// TIA Portal V17 export
// export: Created 2025-03-07T09:17:41.1977773Z, ExportSetting WithDefaults, DisplayName Totally Integrated Automation Portal, DisplayVersion V17 Update 8, DisplayName TIA Portal Openness, DisplayVersion V17 Update 8, DisplayName TIA Portal Version Control Interface, DisplayVersion V17, DisplayName SINAMICS Startdrive Advanced, DisplayVersion V17 SP2, DisplayName SINAMICS Startdrive G110M, G120, G120C, G120D, G120P, G115D, DisplayVersion V17 SP2, DisplayName SINAMICS Startdrive G130, G150, S120, S150, SINAMICS MV, S210, DisplayVersion V17 SP2, DisplayName STEP 7 Professional, DisplayVersion V17 Update 8, DisplayName SINUMERIK ONE STEP 7 Toolbox, DisplayVersion V17 Update 12, DisplayName SINUMERIK 840D sl STEP 7 Toolbox, DisplayVersion V17 Update 12, DisplayName STEP 7 Safety, DisplayVersion V17 Update 6, DisplayName WinCC Advanced, DisplayVersion V17 Update 8
FUNCTION "FC2027_INCREMENTAL_MODE_MG2" : Void   // FC2027, LAD
{ S7_Optimized_Access := 'FALSE' }
AUTHOR : ETXETAR
VERSION : 1.0
// stored: AutoNumber false, IsIECCheckEnabled false, SetENOAutomatically false, UDAEnableTagReadback false
   VAR CONSTANT
      FC_NUMBER : DInt := 2027;
   END_VAR
   VAR_TEMP   // added for the SCL form of the ladder/FBD networks
      _w1 : Bool;
      _w2 : Bool;
   END_VAR
BEGIN

REGION Network 1: GENERAL CONDITIONS
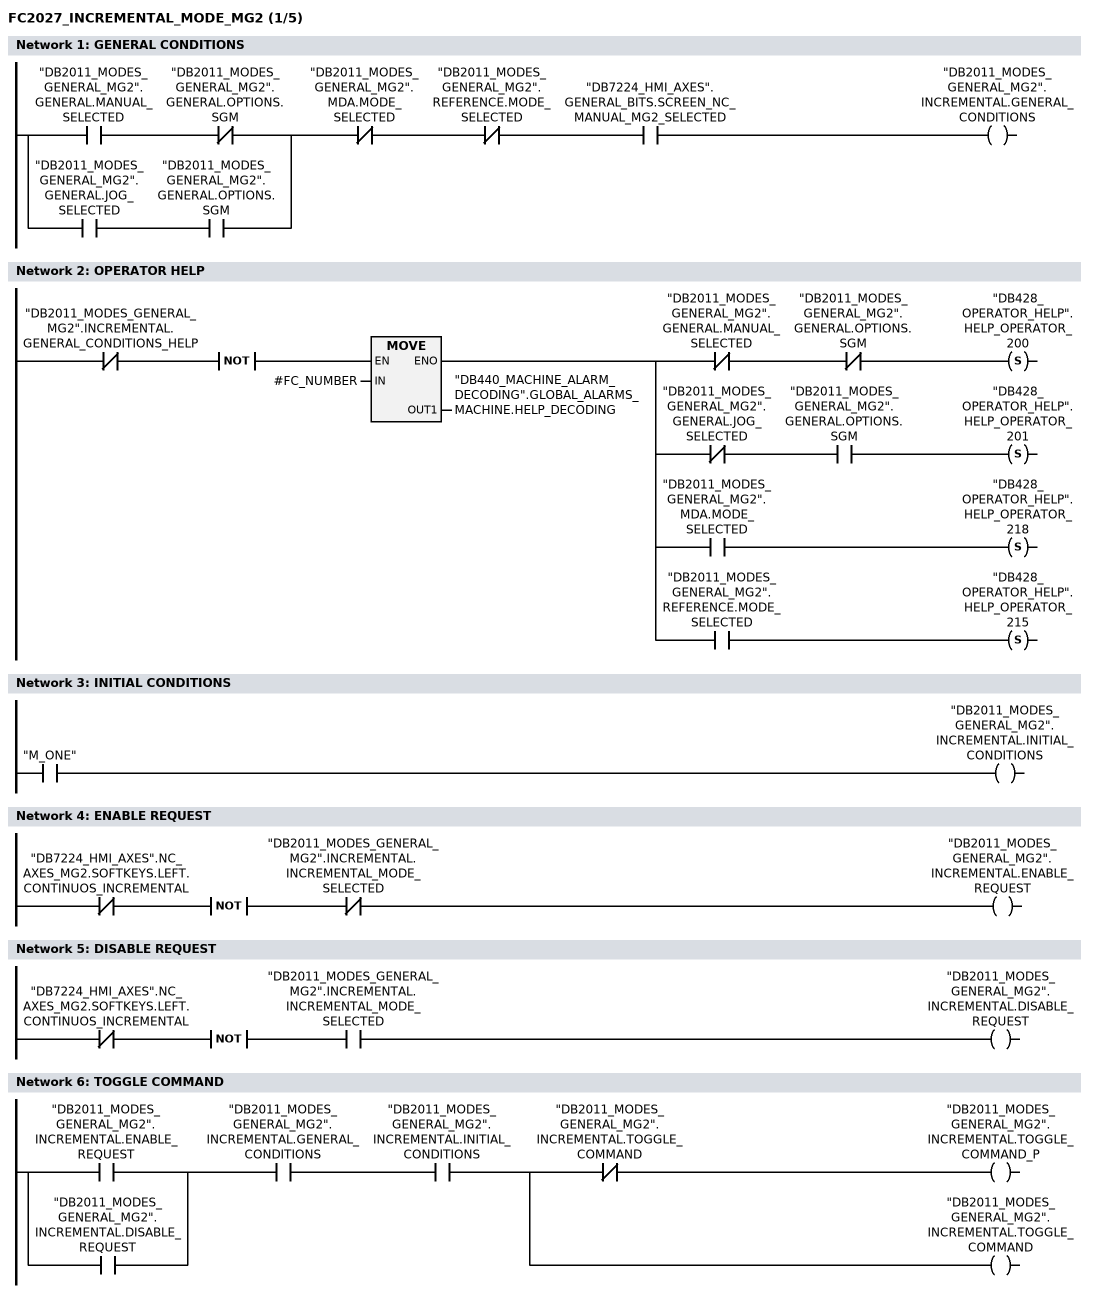
   RUNG wire#powerrail
      Contact( "DB2011_MODES_GENERAL_MG2".GENERAL.MANUAL_SELECTED )
      I_Contact( "DB2011_MODES_GENERAL_MG2".GENERAL.OPTIONS.SGM )
      wire#w1
      I_Contact( "DB2011_MODES_GENERAL_MG2".MDA.MODE_SELECTED )
      I_Contact( "DB2011_MODES_GENERAL_MG2".REFERENCE.MODE_SELECTED )
      Contact( "DB7224_HMI_AXES".GENERAL_BITS.SCREEN_NC_MANUAL_MG2_SELECTED )
      Coil( "DB2011_MODES_GENERAL_MG2".INCREMENTAL.GENERAL_CONDITIONS )
   END_RUNG
   RUNG wire#powerrail
      Contact( "DB2011_MODES_GENERAL_MG2".GENERAL.JOG_SELECTED )
      Contact( "DB2011_MODES_GENERAL_MG2".GENERAL.OPTIONS.SGM )
   END_RUNG wire#w1
   // the same network as SCL:
   "DB2011_MODES_GENERAL_MG2".INCREMENTAL.GENERAL_CONDITIONS := (("DB2011_MODES_GENERAL_MG2".GENERAL.MANUAL_SELECTED AND NOT "DB2011_MODES_GENERAL_MG2".GENERAL.OPTIONS.SGM) OR ("DB2011_MODES_GENERAL_MG2".GENERAL.JOG_SELECTED AND "DB2011_MODES_GENERAL_MG2".GENERAL.OPTIONS.SGM)) AND NOT "DB2011_MODES_GENERAL_MG2".MDA.MODE_SELECTED AND NOT "DB2011_MODES_GENERAL_MG2".REFERENCE.MODE_SELECTED AND "DB7224_HMI_AXES".GENERAL_BITS.SCREEN_NC_MANUAL_MG2_SELECTED;
END_REGION

REGION Network 2: OPERATOR HELP
   RUNG wire#powerrail
      I_Contact( "DB2011_MODES_GENERAL_MG2".INCREMENTAL.GENERAL_CONDITIONS_HELP )
      Not()
      { S7_GenerateENO := "TRUE" } Move(in := #FC_NUMBER, out1 => "DB440_MACHINE_ALARM_DECODING".GLOBAL_ALARMS_MACHINE.HELP_DECODING)
      wire#w1
      I_Contact( "DB2011_MODES_GENERAL_MG2".GENERAL.MANUAL_SELECTED )
      I_Contact( "DB2011_MODES_GENERAL_MG2".GENERAL.OPTIONS.SGM )
      S_Coil( "DB428_OPERATOR_HELP".HELP_OPERATOR_200 )
   END_RUNG
   RUNG wire#w1
      I_Contact( "DB2011_MODES_GENERAL_MG2".GENERAL.JOG_SELECTED )
      Contact( "DB2011_MODES_GENERAL_MG2".GENERAL.OPTIONS.SGM )
      S_Coil( "DB428_OPERATOR_HELP".HELP_OPERATOR_201 )
   END_RUNG
   RUNG wire#w1
      Contact( "DB2011_MODES_GENERAL_MG2".MDA.MODE_SELECTED )
      S_Coil( "DB428_OPERATOR_HELP".HELP_OPERATOR_218 )
   END_RUNG
   RUNG wire#w1
      Contact( "DB2011_MODES_GENERAL_MG2".REFERENCE.MODE_SELECTED )
      S_Coil( "DB428_OPERATOR_HELP".HELP_OPERATOR_215 )
   END_RUNG
   // the same network as SCL:
   // ENO of a box is taken as its EN; it also drops when the box reports an error
   #_w1 := NOT (NOT "DB2011_MODES_GENERAL_MG2".INCREMENTAL.GENERAL_CONDITIONS_HELP);
   IF #_w1 THEN "DB440_MACHINE_ALARM_DECODING".GLOBAL_ALARMS_MACHINE.HELP_DECODING := #FC_NUMBER; END_IF;
   IF #_w1 AND NOT "DB2011_MODES_GENERAL_MG2".GENERAL.MANUAL_SELECTED AND NOT "DB2011_MODES_GENERAL_MG2".GENERAL.OPTIONS.SGM THEN
       "DB428_OPERATOR_HELP".HELP_OPERATOR_200 := TRUE;
   END_IF;
   IF #_w1 AND NOT "DB2011_MODES_GENERAL_MG2".GENERAL.JOG_SELECTED AND "DB2011_MODES_GENERAL_MG2".GENERAL.OPTIONS.SGM THEN
       "DB428_OPERATOR_HELP".HELP_OPERATOR_201 := TRUE;
   END_IF;
   IF #_w1 AND "DB2011_MODES_GENERAL_MG2".MDA.MODE_SELECTED THEN
       "DB428_OPERATOR_HELP".HELP_OPERATOR_218 := TRUE;
   END_IF;
   IF #_w1 AND "DB2011_MODES_GENERAL_MG2".REFERENCE.MODE_SELECTED THEN
       "DB428_OPERATOR_HELP".HELP_OPERATOR_215 := TRUE;
   END_IF;
END_REGION

REGION Network 3: INITIAL CONDITIONS
   RUNG wire#powerrail
      Contact( "M_ONE" )
      Coil( "DB2011_MODES_GENERAL_MG2".INCREMENTAL.INITIAL_CONDITIONS )
   END_RUNG
   // the same network as SCL:
   "DB2011_MODES_GENERAL_MG2".INCREMENTAL.INITIAL_CONDITIONS := "M_ONE";
END_REGION

REGION Network 4: ENABLE REQUEST
   RUNG wire#powerrail
      I_Contact( "DB7224_HMI_AXES".NC_AXES_MG2.SOFTKEYS.LEFT.CONTINUOS_INCREMENTAL )
      Not()
      I_Contact( "DB2011_MODES_GENERAL_MG2".INCREMENTAL.INCREMENTAL_MODE_SELECTED )
      Coil( "DB2011_MODES_GENERAL_MG2".INCREMENTAL.ENABLE_REQUEST )
   END_RUNG
   // the same network as SCL:
   "DB2011_MODES_GENERAL_MG2".INCREMENTAL.ENABLE_REQUEST := NOT (NOT "DB7224_HMI_AXES".NC_AXES_MG2.SOFTKEYS.LEFT.CONTINUOS_INCREMENTAL) AND NOT "DB2011_MODES_GENERAL_MG2".INCREMENTAL.INCREMENTAL_MODE_SELECTED;
END_REGION

REGION Network 5: DISABLE REQUEST
   RUNG wire#powerrail
      I_Contact( "DB7224_HMI_AXES".NC_AXES_MG2.SOFTKEYS.LEFT.CONTINUOS_INCREMENTAL )
      Not()
      Contact( "DB2011_MODES_GENERAL_MG2".INCREMENTAL.INCREMENTAL_MODE_SELECTED )
      Coil( "DB2011_MODES_GENERAL_MG2".INCREMENTAL.DISABLE_REQUEST )
   END_RUNG
   // the same network as SCL:
   "DB2011_MODES_GENERAL_MG2".INCREMENTAL.DISABLE_REQUEST := NOT (NOT "DB7224_HMI_AXES".NC_AXES_MG2.SOFTKEYS.LEFT.CONTINUOS_INCREMENTAL) AND "DB2011_MODES_GENERAL_MG2".INCREMENTAL.INCREMENTAL_MODE_SELECTED;
END_REGION

REGION Network 6: TOGGLE COMMAND
   RUNG wire#powerrail
      Contact( "DB2011_MODES_GENERAL_MG2".INCREMENTAL.ENABLE_REQUEST )
      wire#w1
      Contact( "DB2011_MODES_GENERAL_MG2".INCREMENTAL.GENERAL_CONDITIONS )
      Contact( "DB2011_MODES_GENERAL_MG2".INCREMENTAL.INITIAL_CONDITIONS )
      wire#w2
      I_Contact( "DB2011_MODES_GENERAL_MG2".INCREMENTAL.TOGGLE_COMMAND )
      Coil( "DB2011_MODES_GENERAL_MG2".INCREMENTAL.TOGGLE_COMMAND_P )
   END_RUNG
   RUNG wire#powerrail
      Contact( "DB2011_MODES_GENERAL_MG2".INCREMENTAL.DISABLE_REQUEST )
   END_RUNG wire#w1
   RUNG wire#w2
      Coil( "DB2011_MODES_GENERAL_MG2".INCREMENTAL.TOGGLE_COMMAND )
   END_RUNG
   // the same network as SCL:
   #_w1 := ("DB2011_MODES_GENERAL_MG2".INCREMENTAL.ENABLE_REQUEST OR "DB2011_MODES_GENERAL_MG2".INCREMENTAL.DISABLE_REQUEST) AND "DB2011_MODES_GENERAL_MG2".INCREMENTAL.GENERAL_CONDITIONS AND "DB2011_MODES_GENERAL_MG2".INCREMENTAL.INITIAL_CONDITIONS;
   "DB2011_MODES_GENERAL_MG2".INCREMENTAL.TOGGLE_COMMAND_P := #_w1 AND NOT "DB2011_MODES_GENERAL_MG2".INCREMENTAL.TOGGLE_COMMAND;
   "DB2011_MODES_GENERAL_MG2".INCREMENTAL.TOGGLE_COMMAND := #_w1;
END_REGION

REGION Network 7: INCREMENTAL MODE SELECTED
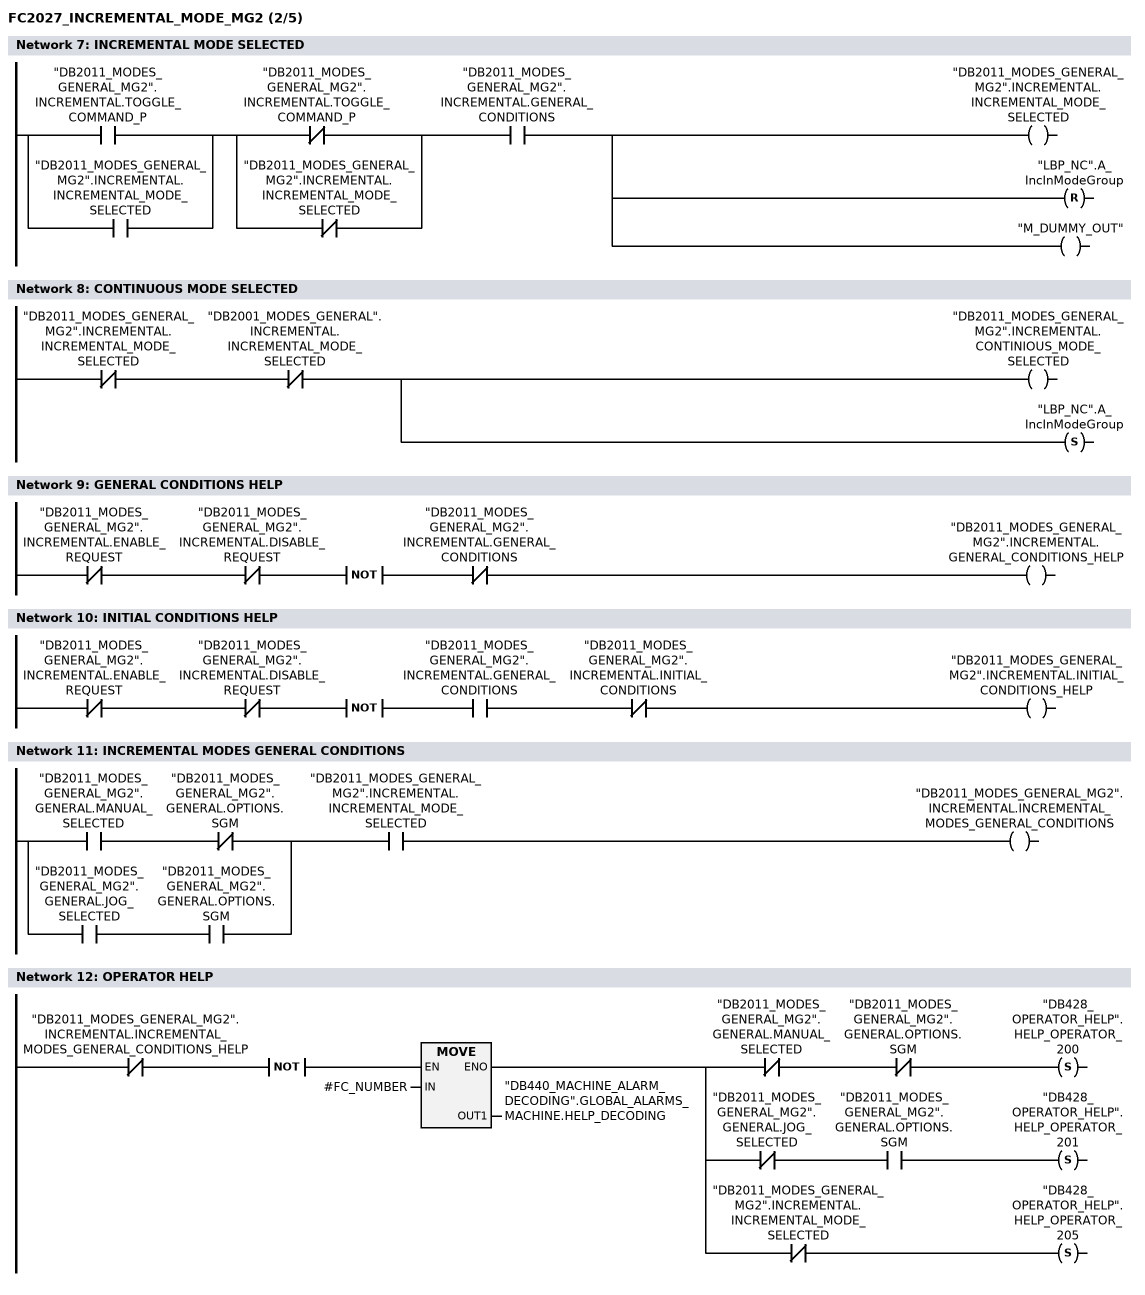
   RUNG wire#powerrail
      Contact( "DB2011_MODES_GENERAL_MG2".INCREMENTAL.TOGGLE_COMMAND_P )
      wire#w1
      I_Contact( "DB2011_MODES_GENERAL_MG2".INCREMENTAL.TOGGLE_COMMAND_P )
      wire#w2
      Contact( "DB2011_MODES_GENERAL_MG2".INCREMENTAL.GENERAL_CONDITIONS )
      wire#w3
      Coil( "DB2011_MODES_GENERAL_MG2".INCREMENTAL.INCREMENTAL_MODE_SELECTED )
   END_RUNG
   RUNG wire#powerrail
      Contact( "DB2011_MODES_GENERAL_MG2".INCREMENTAL.INCREMENTAL_MODE_SELECTED )
   END_RUNG wire#w1
   RUNG wire#w1
      I_Contact( "DB2011_MODES_GENERAL_MG2".INCREMENTAL.INCREMENTAL_MODE_SELECTED )
   END_RUNG wire#w2
   RUNG wire#w3
      R_Coil( "LBP_NC".A_IncInModeGroup )
   END_RUNG
   RUNG wire#w3
      Coil( "M_DUMMY_OUT" )
   END_RUNG
   // the same network as SCL:
   "DB2011_MODES_GENERAL_MG2".INCREMENTAL.INCREMENTAL_MODE_SELECTED := ("DB2011_MODES_GENERAL_MG2".INCREMENTAL.TOGGLE_COMMAND_P OR "DB2011_MODES_GENERAL_MG2".INCREMENTAL.INCREMENTAL_MODE_SELECTED) AND (NOT "DB2011_MODES_GENERAL_MG2".INCREMENTAL.TOGGLE_COMMAND_P OR NOT "DB2011_MODES_GENERAL_MG2".INCREMENTAL.INCREMENTAL_MODE_SELECTED) AND "DB2011_MODES_GENERAL_MG2".INCREMENTAL.GENERAL_CONDITIONS;
   IF "DB2011_MODES_GENERAL_MG2".INCREMENTAL.INCREMENTAL_MODE_SELECTED THEN
       "LBP_NC".A_IncInModeGroup := FALSE;
   END_IF;
   "M_DUMMY_OUT" := "DB2011_MODES_GENERAL_MG2".INCREMENTAL.INCREMENTAL_MODE_SELECTED;
END_REGION

REGION Network 8: CONTINUOUS MODE SELECTED
   RUNG wire#powerrail
      I_Contact( "DB2011_MODES_GENERAL_MG2".INCREMENTAL.INCREMENTAL_MODE_SELECTED )
      I_Contact( "DB2001_MODES_GENERAL".INCREMENTAL.INCREMENTAL_MODE_SELECTED )
      wire#w1
      Coil( "DB2011_MODES_GENERAL_MG2".INCREMENTAL.CONTINIOUS_MODE_SELECTED )
   END_RUNG
   RUNG wire#w1
      S_Coil( "LBP_NC".A_IncInModeGroup )
   END_RUNG
   // the same network as SCL:
   "DB2011_MODES_GENERAL_MG2".INCREMENTAL.CONTINIOUS_MODE_SELECTED := NOT "DB2011_MODES_GENERAL_MG2".INCREMENTAL.INCREMENTAL_MODE_SELECTED AND NOT "DB2001_MODES_GENERAL".INCREMENTAL.INCREMENTAL_MODE_SELECTED;
   IF "DB2011_MODES_GENERAL_MG2".INCREMENTAL.CONTINIOUS_MODE_SELECTED THEN
       "LBP_NC".A_IncInModeGroup := TRUE;
   END_IF;
END_REGION

REGION Network 9: GENERAL CONDITIONS HELP
   RUNG wire#powerrail
      I_Contact( "DB2011_MODES_GENERAL_MG2".INCREMENTAL.ENABLE_REQUEST )
      I_Contact( "DB2011_MODES_GENERAL_MG2".INCREMENTAL.DISABLE_REQUEST )
      Not()
      I_Contact( "DB2011_MODES_GENERAL_MG2".INCREMENTAL.GENERAL_CONDITIONS )
      Coil( "DB2011_MODES_GENERAL_MG2".INCREMENTAL.GENERAL_CONDITIONS_HELP )
   END_RUNG
   // the same network as SCL:
   "DB2011_MODES_GENERAL_MG2".INCREMENTAL.GENERAL_CONDITIONS_HELP := NOT (NOT "DB2011_MODES_GENERAL_MG2".INCREMENTAL.ENABLE_REQUEST AND NOT "DB2011_MODES_GENERAL_MG2".INCREMENTAL.DISABLE_REQUEST) AND NOT "DB2011_MODES_GENERAL_MG2".INCREMENTAL.GENERAL_CONDITIONS;
END_REGION

REGION Network 10: INITIAL CONDITIONS HELP
   RUNG wire#powerrail
      I_Contact( "DB2011_MODES_GENERAL_MG2".INCREMENTAL.ENABLE_REQUEST )
      I_Contact( "DB2011_MODES_GENERAL_MG2".INCREMENTAL.DISABLE_REQUEST )
      Not()
      Contact( "DB2011_MODES_GENERAL_MG2".INCREMENTAL.GENERAL_CONDITIONS )
      I_Contact( "DB2011_MODES_GENERAL_MG2".INCREMENTAL.INITIAL_CONDITIONS )
      Coil( "DB2011_MODES_GENERAL_MG2".INCREMENTAL.INITIAL_CONDITIONS_HELP )
   END_RUNG
   // the same network as SCL:
   "DB2011_MODES_GENERAL_MG2".INCREMENTAL.INITIAL_CONDITIONS_HELP := NOT (NOT "DB2011_MODES_GENERAL_MG2".INCREMENTAL.ENABLE_REQUEST AND NOT "DB2011_MODES_GENERAL_MG2".INCREMENTAL.DISABLE_REQUEST) AND "DB2011_MODES_GENERAL_MG2".INCREMENTAL.GENERAL_CONDITIONS AND NOT "DB2011_MODES_GENERAL_MG2".INCREMENTAL.INITIAL_CONDITIONS;
END_REGION

REGION Network 11: INCREMENTAL MODES GENERAL CONDITIONS
   RUNG wire#powerrail
      Contact( "DB2011_MODES_GENERAL_MG2".GENERAL.MANUAL_SELECTED )
      I_Contact( "DB2011_MODES_GENERAL_MG2".GENERAL.OPTIONS.SGM )
      wire#w1
      Contact( "DB2011_MODES_GENERAL_MG2".INCREMENTAL.INCREMENTAL_MODE_SELECTED )
      Coil( "DB2011_MODES_GENERAL_MG2".INCREMENTAL.INCREMENTAL_MODES_GENERAL_CONDITIONS )
   END_RUNG
   RUNG wire#powerrail
      Contact( "DB2011_MODES_GENERAL_MG2".GENERAL.JOG_SELECTED )
      Contact( "DB2011_MODES_GENERAL_MG2".GENERAL.OPTIONS.SGM )
   END_RUNG wire#w1
   // the same network as SCL:
   "DB2011_MODES_GENERAL_MG2".INCREMENTAL.INCREMENTAL_MODES_GENERAL_CONDITIONS := (("DB2011_MODES_GENERAL_MG2".GENERAL.MANUAL_SELECTED AND NOT "DB2011_MODES_GENERAL_MG2".GENERAL.OPTIONS.SGM) OR ("DB2011_MODES_GENERAL_MG2".GENERAL.JOG_SELECTED AND "DB2011_MODES_GENERAL_MG2".GENERAL.OPTIONS.SGM)) AND "DB2011_MODES_GENERAL_MG2".INCREMENTAL.INCREMENTAL_MODE_SELECTED;
END_REGION

REGION Network 12: OPERATOR HELP
   RUNG wire#powerrail
      I_Contact( "DB2011_MODES_GENERAL_MG2".INCREMENTAL.INCREMENTAL_MODES_GENERAL_CONDITIONS_HELP )
      Not()
      { S7_GenerateENO := "TRUE" } Move(in := #FC_NUMBER, out1 => "DB440_MACHINE_ALARM_DECODING".GLOBAL_ALARMS_MACHINE.HELP_DECODING)
      wire#w1
      I_Contact( "DB2011_MODES_GENERAL_MG2".GENERAL.MANUAL_SELECTED )
      I_Contact( "DB2011_MODES_GENERAL_MG2".GENERAL.OPTIONS.SGM )
      S_Coil( "DB428_OPERATOR_HELP".HELP_OPERATOR_200 )
   END_RUNG
   RUNG wire#w1
      I_Contact( "DB2011_MODES_GENERAL_MG2".GENERAL.JOG_SELECTED )
      Contact( "DB2011_MODES_GENERAL_MG2".GENERAL.OPTIONS.SGM )
      S_Coil( "DB428_OPERATOR_HELP".HELP_OPERATOR_201 )
   END_RUNG
   RUNG wire#w1
      I_Contact( "DB2011_MODES_GENERAL_MG2".INCREMENTAL.INCREMENTAL_MODE_SELECTED )
      S_Coil( "DB428_OPERATOR_HELP".HELP_OPERATOR_205 )
   END_RUNG
   // the same network as SCL:
   // ENO of a box is taken as its EN; it also drops when the box reports an error
   #_w1 := NOT (NOT "DB2011_MODES_GENERAL_MG2".INCREMENTAL.INCREMENTAL_MODES_GENERAL_CONDITIONS_HELP);
   IF #_w1 THEN "DB440_MACHINE_ALARM_DECODING".GLOBAL_ALARMS_MACHINE.HELP_DECODING := #FC_NUMBER; END_IF;
   IF #_w1 AND NOT "DB2011_MODES_GENERAL_MG2".GENERAL.MANUAL_SELECTED AND NOT "DB2011_MODES_GENERAL_MG2".GENERAL.OPTIONS.SGM THEN
       "DB428_OPERATOR_HELP".HELP_OPERATOR_200 := TRUE;
   END_IF;
   IF #_w1 AND NOT "DB2011_MODES_GENERAL_MG2".GENERAL.JOG_SELECTED AND "DB2011_MODES_GENERAL_MG2".GENERAL.OPTIONS.SGM THEN
       "DB428_OPERATOR_HELP".HELP_OPERATOR_201 := TRUE;
   END_IF;
   IF #_w1 AND NOT "DB2011_MODES_GENERAL_MG2".INCREMENTAL.INCREMENTAL_MODE_SELECTED THEN
       "DB428_OPERATOR_HELP".HELP_OPERATOR_205 := TRUE;
   END_IF;
END_REGION

REGION Network 13: INCREMENTAL MODES INITIAL CONDITIONS
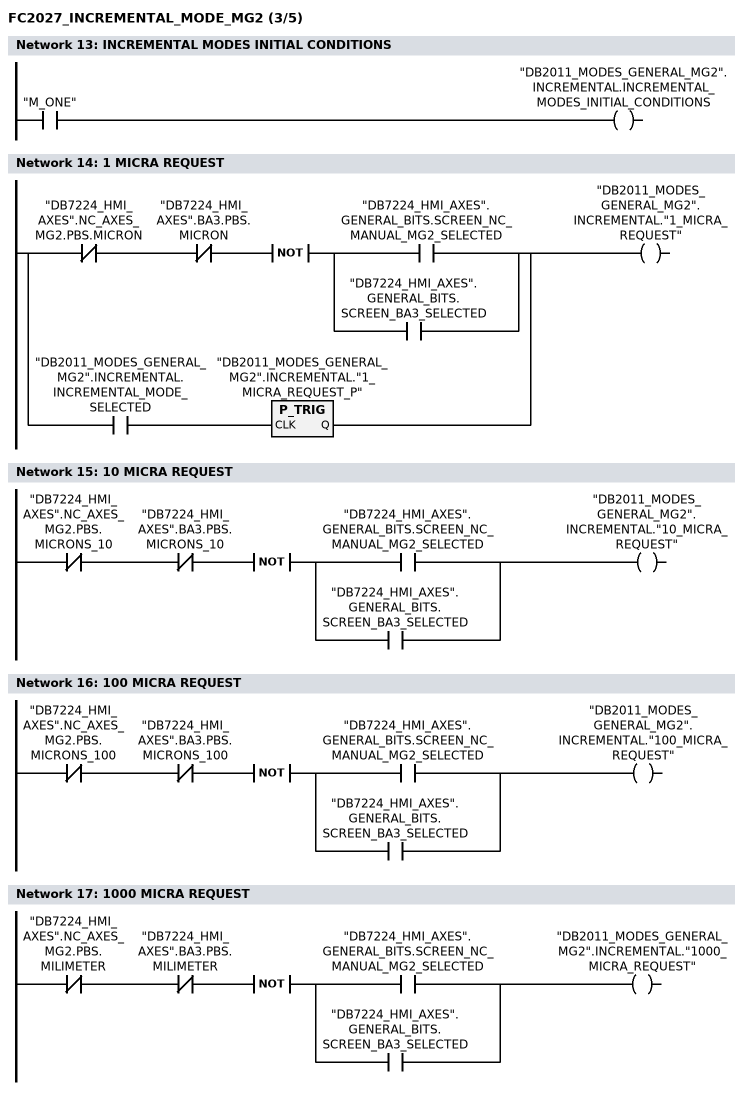
   RUNG wire#powerrail
      Contact( "M_ONE" )
      Coil( "DB2011_MODES_GENERAL_MG2".INCREMENTAL.INCREMENTAL_MODES_INITIAL_CONDITIONS )
   END_RUNG
   // the same network as SCL:
   "DB2011_MODES_GENERAL_MG2".INCREMENTAL.INCREMENTAL_MODES_INITIAL_CONDITIONS := "M_ONE";
END_REGION

REGION Network 14: 1 MICRA REQUEST
   RUNG wire#powerrail
      I_Contact( "DB7224_HMI_AXES".NC_AXES_MG2.PBS.MICRON )
      I_Contact( "DB7224_HMI_AXES".BA3.PBS.MICRON )
      Not()
      wire#w1
      Contact( "DB7224_HMI_AXES".GENERAL_BITS.SCREEN_NC_MANUAL_MG2_SELECTED )
      wire#w2
      Coil( "DB2011_MODES_GENERAL_MG2".INCREMENTAL."1_MICRA_REQUEST" )
   END_RUNG
   RUNG wire#w1
      Contact( "DB7224_HMI_AXES".GENERAL_BITS.SCREEN_BA3_SELECTED )
   END_RUNG wire#w2
   RUNG wire#powerrail
      Contact( "DB2011_MODES_GENERAL_MG2".INCREMENTAL.INCREMENTAL_MODE_SELECTED )
      P_Trig( "DB2011_MODES_GENERAL_MG2".INCREMENTAL."1_MICRA_REQUEST_P" )
   END_RUNG wire#w2
   // the same network as SCL:
   #_w1 := "DB2011_MODES_GENERAL_MG2".INCREMENTAL.INCREMENTAL_MODE_SELECTED AND NOT "DB2011_MODES_GENERAL_MG2".INCREMENTAL."1_MICRA_REQUEST_P";   // rising edge
   "DB2011_MODES_GENERAL_MG2".INCREMENTAL."1_MICRA_REQUEST_P" := "DB2011_MODES_GENERAL_MG2".INCREMENTAL.INCREMENTAL_MODE_SELECTED;
   "DB2011_MODES_GENERAL_MG2".INCREMENTAL."1_MICRA_REQUEST" := (NOT (NOT "DB7224_HMI_AXES".NC_AXES_MG2.PBS.MICRON AND NOT "DB7224_HMI_AXES".BA3.PBS.MICRON) AND ("DB7224_HMI_AXES".GENERAL_BITS.SCREEN_NC_MANUAL_MG2_SELECTED OR "DB7224_HMI_AXES".GENERAL_BITS.SCREEN_BA3_SELECTED)) OR #_w1;
END_REGION

REGION Network 15: 10 MICRA REQUEST
   RUNG wire#powerrail
      I_Contact( "DB7224_HMI_AXES".NC_AXES_MG2.PBS.MICRONS_10 )
      I_Contact( "DB7224_HMI_AXES".BA3.PBS.MICRONS_10 )
      Not()
      wire#w1
      Contact( "DB7224_HMI_AXES".GENERAL_BITS.SCREEN_NC_MANUAL_MG2_SELECTED )
      wire#w2
      Coil( "DB2011_MODES_GENERAL_MG2".INCREMENTAL."10_MICRA_REQUEST" )
   END_RUNG
   RUNG wire#w1
      Contact( "DB7224_HMI_AXES".GENERAL_BITS.SCREEN_BA3_SELECTED )
   END_RUNG wire#w2
   // the same network as SCL:
   "DB2011_MODES_GENERAL_MG2".INCREMENTAL."10_MICRA_REQUEST" := NOT (NOT "DB7224_HMI_AXES".NC_AXES_MG2.PBS.MICRONS_10 AND NOT "DB7224_HMI_AXES".BA3.PBS.MICRONS_10) AND ("DB7224_HMI_AXES".GENERAL_BITS.SCREEN_NC_MANUAL_MG2_SELECTED OR "DB7224_HMI_AXES".GENERAL_BITS.SCREEN_BA3_SELECTED);
END_REGION

REGION Network 16: 100 MICRA REQUEST
   RUNG wire#powerrail
      I_Contact( "DB7224_HMI_AXES".NC_AXES_MG2.PBS.MICRONS_100 )
      I_Contact( "DB7224_HMI_AXES".BA3.PBS.MICRONS_100 )
      Not()
      wire#w1
      Contact( "DB7224_HMI_AXES".GENERAL_BITS.SCREEN_NC_MANUAL_MG2_SELECTED )
      wire#w2
      Coil( "DB2011_MODES_GENERAL_MG2".INCREMENTAL."100_MICRA_REQUEST" )
   END_RUNG
   RUNG wire#w1
      Contact( "DB7224_HMI_AXES".GENERAL_BITS.SCREEN_BA3_SELECTED )
   END_RUNG wire#w2
   // the same network as SCL:
   "DB2011_MODES_GENERAL_MG2".INCREMENTAL."100_MICRA_REQUEST" := NOT (NOT "DB7224_HMI_AXES".NC_AXES_MG2.PBS.MICRONS_100 AND NOT "DB7224_HMI_AXES".BA3.PBS.MICRONS_100) AND ("DB7224_HMI_AXES".GENERAL_BITS.SCREEN_NC_MANUAL_MG2_SELECTED OR "DB7224_HMI_AXES".GENERAL_BITS.SCREEN_BA3_SELECTED);
END_REGION

REGION Network 17: 1000 MICRA REQUEST
   RUNG wire#powerrail
      I_Contact( "DB7224_HMI_AXES".NC_AXES_MG2.PBS.MILIMETER )
      I_Contact( "DB7224_HMI_AXES".BA3.PBS.MILIMETER )
      Not()
      wire#w1
      Contact( "DB7224_HMI_AXES".GENERAL_BITS.SCREEN_NC_MANUAL_MG2_SELECTED )
      wire#w2
      Coil( "DB2011_MODES_GENERAL_MG2".INCREMENTAL."1000_MICRA_REQUEST" )
   END_RUNG
   RUNG wire#w1
      Contact( "DB7224_HMI_AXES".GENERAL_BITS.SCREEN_BA3_SELECTED )
   END_RUNG wire#w2
   // the same network as SCL:
   "DB2011_MODES_GENERAL_MG2".INCREMENTAL."1000_MICRA_REQUEST" := NOT (NOT "DB7224_HMI_AXES".NC_AXES_MG2.PBS.MILIMETER AND NOT "DB7224_HMI_AXES".BA3.PBS.MILIMETER) AND ("DB7224_HMI_AXES".GENERAL_BITS.SCREEN_NC_MANUAL_MG2_SELECTED OR "DB7224_HMI_AXES".GENERAL_BITS.SCREEN_BA3_SELECTED);
END_REGION

REGION Network 18: 1 MICRA SELECTED
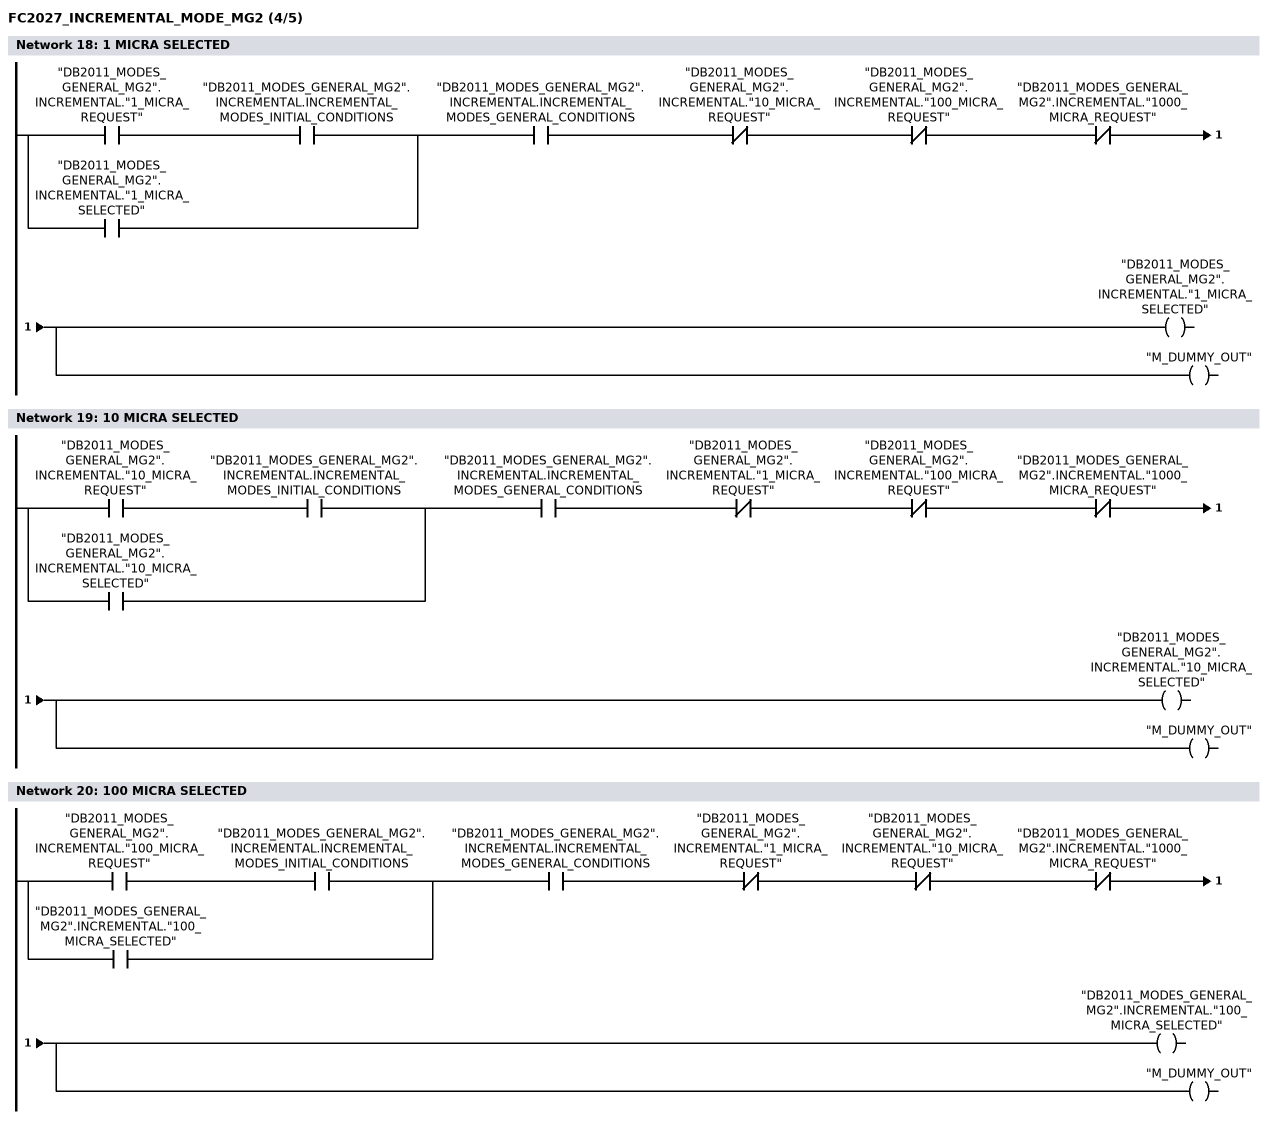
   RUNG wire#powerrail
      Contact( "DB2011_MODES_GENERAL_MG2".INCREMENTAL."1_MICRA_REQUEST" )
      Contact( "DB2011_MODES_GENERAL_MG2".INCREMENTAL.INCREMENTAL_MODES_INITIAL_CONDITIONS )
      wire#w1
      Contact( "DB2011_MODES_GENERAL_MG2".INCREMENTAL.INCREMENTAL_MODES_GENERAL_CONDITIONS )
      I_Contact( "DB2011_MODES_GENERAL_MG2".INCREMENTAL."10_MICRA_REQUEST" )
      I_Contact( "DB2011_MODES_GENERAL_MG2".INCREMENTAL."100_MICRA_REQUEST" )
      I_Contact( "DB2011_MODES_GENERAL_MG2".INCREMENTAL."1000_MICRA_REQUEST" )
      wire#w2
      Coil( "DB2011_MODES_GENERAL_MG2".INCREMENTAL."1_MICRA_SELECTED" )
   END_RUNG
   RUNG wire#powerrail
      Contact( "DB2011_MODES_GENERAL_MG2".INCREMENTAL."1_MICRA_SELECTED" )
   END_RUNG wire#w1
   RUNG wire#w2
      Coil( "M_DUMMY_OUT" )
   END_RUNG
   // the same network as SCL:
   "DB2011_MODES_GENERAL_MG2".INCREMENTAL."1_MICRA_SELECTED" := (("DB2011_MODES_GENERAL_MG2".INCREMENTAL."1_MICRA_REQUEST" AND "DB2011_MODES_GENERAL_MG2".INCREMENTAL.INCREMENTAL_MODES_INITIAL_CONDITIONS) OR "DB2011_MODES_GENERAL_MG2".INCREMENTAL."1_MICRA_SELECTED") AND "DB2011_MODES_GENERAL_MG2".INCREMENTAL.INCREMENTAL_MODES_GENERAL_CONDITIONS AND NOT "DB2011_MODES_GENERAL_MG2".INCREMENTAL."10_MICRA_REQUEST" AND NOT "DB2011_MODES_GENERAL_MG2".INCREMENTAL."100_MICRA_REQUEST" AND NOT "DB2011_MODES_GENERAL_MG2".INCREMENTAL."1000_MICRA_REQUEST";
   "M_DUMMY_OUT" := "DB2011_MODES_GENERAL_MG2".INCREMENTAL."1_MICRA_SELECTED";
END_REGION

REGION Network 19: 10 MICRA SELECTED
   RUNG wire#powerrail
      Contact( "DB2011_MODES_GENERAL_MG2".INCREMENTAL."10_MICRA_REQUEST" )
      Contact( "DB2011_MODES_GENERAL_MG2".INCREMENTAL.INCREMENTAL_MODES_INITIAL_CONDITIONS )
      wire#w1
      Contact( "DB2011_MODES_GENERAL_MG2".INCREMENTAL.INCREMENTAL_MODES_GENERAL_CONDITIONS )
      I_Contact( "DB2011_MODES_GENERAL_MG2".INCREMENTAL."1_MICRA_REQUEST" )
      I_Contact( "DB2011_MODES_GENERAL_MG2".INCREMENTAL."100_MICRA_REQUEST" )
      I_Contact( "DB2011_MODES_GENERAL_MG2".INCREMENTAL."1000_MICRA_REQUEST" )
      wire#w2
      Coil( "DB2011_MODES_GENERAL_MG2".INCREMENTAL."10_MICRA_SELECTED" )
   END_RUNG
   RUNG wire#powerrail
      Contact( "DB2011_MODES_GENERAL_MG2".INCREMENTAL."10_MICRA_SELECTED" )
   END_RUNG wire#w1
   RUNG wire#w2
      Coil( "M_DUMMY_OUT" )
   END_RUNG
   // the same network as SCL:
   "DB2011_MODES_GENERAL_MG2".INCREMENTAL."10_MICRA_SELECTED" := (("DB2011_MODES_GENERAL_MG2".INCREMENTAL."10_MICRA_REQUEST" AND "DB2011_MODES_GENERAL_MG2".INCREMENTAL.INCREMENTAL_MODES_INITIAL_CONDITIONS) OR "DB2011_MODES_GENERAL_MG2".INCREMENTAL."10_MICRA_SELECTED") AND "DB2011_MODES_GENERAL_MG2".INCREMENTAL.INCREMENTAL_MODES_GENERAL_CONDITIONS AND NOT "DB2011_MODES_GENERAL_MG2".INCREMENTAL."1_MICRA_REQUEST" AND NOT "DB2011_MODES_GENERAL_MG2".INCREMENTAL."100_MICRA_REQUEST" AND NOT "DB2011_MODES_GENERAL_MG2".INCREMENTAL."1000_MICRA_REQUEST";
   "M_DUMMY_OUT" := "DB2011_MODES_GENERAL_MG2".INCREMENTAL."10_MICRA_SELECTED";
END_REGION

REGION Network 20: 100 MICRA SELECTED
   RUNG wire#powerrail
      Contact( "DB2011_MODES_GENERAL_MG2".INCREMENTAL."100_MICRA_REQUEST" )
      Contact( "DB2011_MODES_GENERAL_MG2".INCREMENTAL.INCREMENTAL_MODES_INITIAL_CONDITIONS )
      wire#w1
      Contact( "DB2011_MODES_GENERAL_MG2".INCREMENTAL.INCREMENTAL_MODES_GENERAL_CONDITIONS )
      I_Contact( "DB2011_MODES_GENERAL_MG2".INCREMENTAL."1_MICRA_REQUEST" )
      I_Contact( "DB2011_MODES_GENERAL_MG2".INCREMENTAL."10_MICRA_REQUEST" )
      I_Contact( "DB2011_MODES_GENERAL_MG2".INCREMENTAL."1000_MICRA_REQUEST" )
      wire#w2
      Coil( "DB2011_MODES_GENERAL_MG2".INCREMENTAL."100_MICRA_SELECTED" )
   END_RUNG
   RUNG wire#powerrail
      Contact( "DB2011_MODES_GENERAL_MG2".INCREMENTAL."100_MICRA_SELECTED" )
   END_RUNG wire#w1
   RUNG wire#w2
      Coil( "M_DUMMY_OUT" )
   END_RUNG
   // the same network as SCL:
   "DB2011_MODES_GENERAL_MG2".INCREMENTAL."100_MICRA_SELECTED" := (("DB2011_MODES_GENERAL_MG2".INCREMENTAL."100_MICRA_REQUEST" AND "DB2011_MODES_GENERAL_MG2".INCREMENTAL.INCREMENTAL_MODES_INITIAL_CONDITIONS) OR "DB2011_MODES_GENERAL_MG2".INCREMENTAL."100_MICRA_SELECTED") AND "DB2011_MODES_GENERAL_MG2".INCREMENTAL.INCREMENTAL_MODES_GENERAL_CONDITIONS AND NOT "DB2011_MODES_GENERAL_MG2".INCREMENTAL."1_MICRA_REQUEST" AND NOT "DB2011_MODES_GENERAL_MG2".INCREMENTAL."10_MICRA_REQUEST" AND NOT "DB2011_MODES_GENERAL_MG2".INCREMENTAL."1000_MICRA_REQUEST";
   "M_DUMMY_OUT" := "DB2011_MODES_GENERAL_MG2".INCREMENTAL."100_MICRA_SELECTED";
END_REGION

REGION Network 21: 1000 MICRA SELECTED
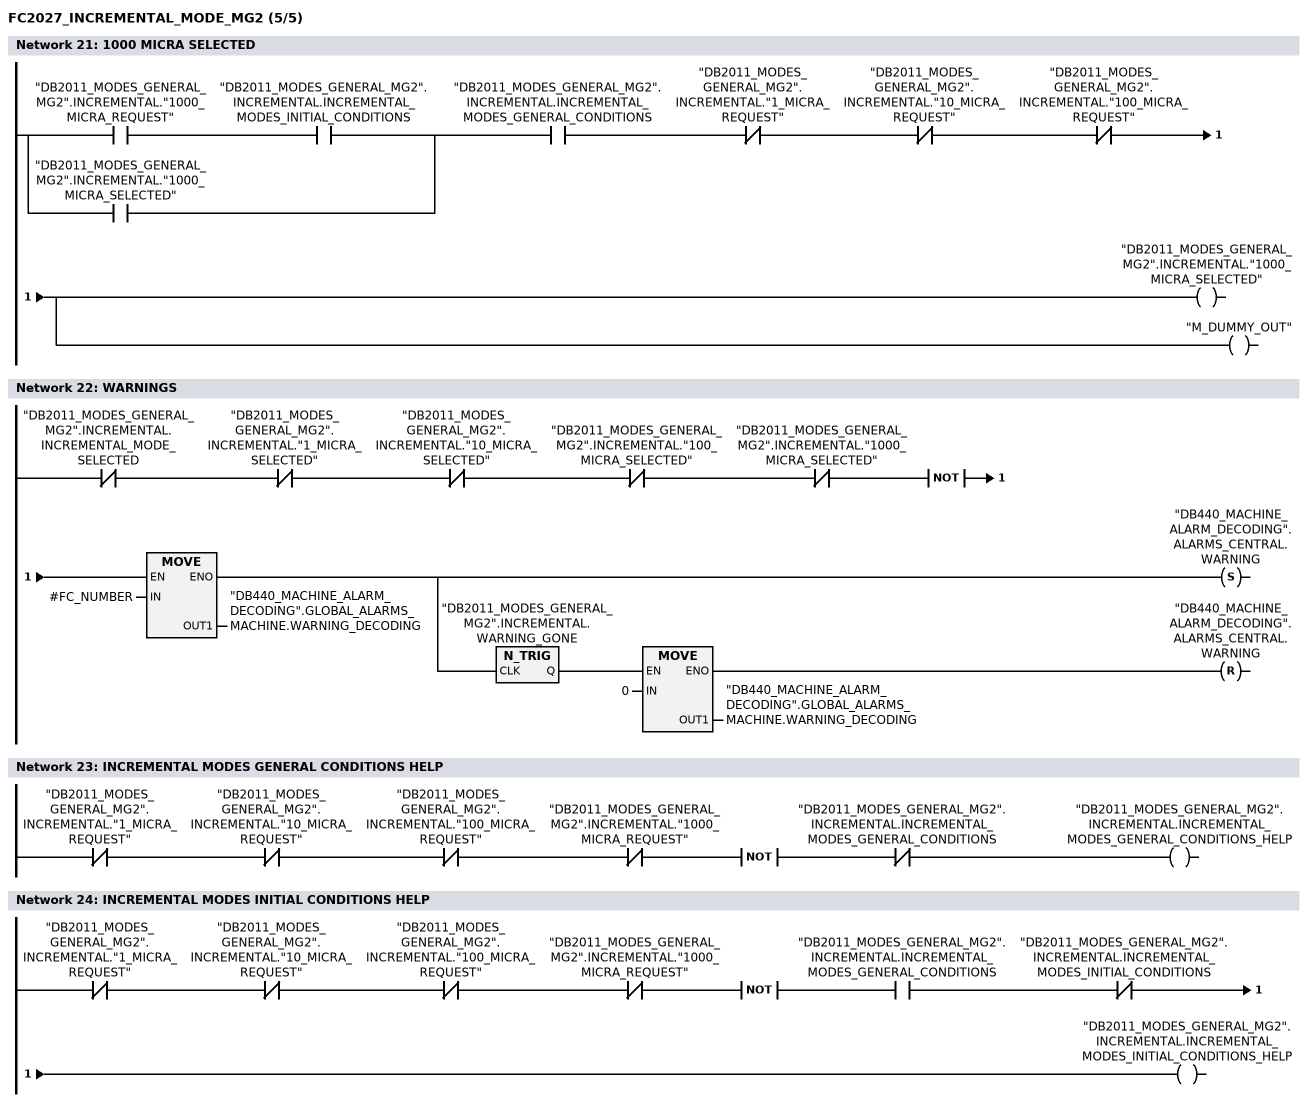
   RUNG wire#powerrail
      Contact( "DB2011_MODES_GENERAL_MG2".INCREMENTAL."1000_MICRA_REQUEST" )
      Contact( "DB2011_MODES_GENERAL_MG2".INCREMENTAL.INCREMENTAL_MODES_INITIAL_CONDITIONS )
      wire#w1
      Contact( "DB2011_MODES_GENERAL_MG2".INCREMENTAL.INCREMENTAL_MODES_GENERAL_CONDITIONS )
      I_Contact( "DB2011_MODES_GENERAL_MG2".INCREMENTAL."1_MICRA_REQUEST" )
      I_Contact( "DB2011_MODES_GENERAL_MG2".INCREMENTAL."10_MICRA_REQUEST" )
      I_Contact( "DB2011_MODES_GENERAL_MG2".INCREMENTAL."100_MICRA_REQUEST" )
      wire#w2
      Coil( "DB2011_MODES_GENERAL_MG2".INCREMENTAL."1000_MICRA_SELECTED" )
   END_RUNG
   RUNG wire#powerrail
      Contact( "DB2011_MODES_GENERAL_MG2".INCREMENTAL."1000_MICRA_SELECTED" )
   END_RUNG wire#w1
   RUNG wire#w2
      Coil( "M_DUMMY_OUT" )
   END_RUNG
   // the same network as SCL:
   "DB2011_MODES_GENERAL_MG2".INCREMENTAL."1000_MICRA_SELECTED" := (("DB2011_MODES_GENERAL_MG2".INCREMENTAL."1000_MICRA_REQUEST" AND "DB2011_MODES_GENERAL_MG2".INCREMENTAL.INCREMENTAL_MODES_INITIAL_CONDITIONS) OR "DB2011_MODES_GENERAL_MG2".INCREMENTAL."1000_MICRA_SELECTED") AND "DB2011_MODES_GENERAL_MG2".INCREMENTAL.INCREMENTAL_MODES_GENERAL_CONDITIONS AND NOT "DB2011_MODES_GENERAL_MG2".INCREMENTAL."1_MICRA_REQUEST" AND NOT "DB2011_MODES_GENERAL_MG2".INCREMENTAL."10_MICRA_REQUEST" AND NOT "DB2011_MODES_GENERAL_MG2".INCREMENTAL."100_MICRA_REQUEST";
   "M_DUMMY_OUT" := "DB2011_MODES_GENERAL_MG2".INCREMENTAL."1000_MICRA_SELECTED";
END_REGION

REGION Network 22: WARNINGS
   RUNG wire#powerrail
      I_Contact( "DB2011_MODES_GENERAL_MG2".INCREMENTAL.INCREMENTAL_MODE_SELECTED )
      I_Contact( "DB2011_MODES_GENERAL_MG2".INCREMENTAL."1_MICRA_SELECTED" )
      I_Contact( "DB2011_MODES_GENERAL_MG2".INCREMENTAL."10_MICRA_SELECTED" )
      I_Contact( "DB2011_MODES_GENERAL_MG2".INCREMENTAL."100_MICRA_SELECTED" )
      I_Contact( "DB2011_MODES_GENERAL_MG2".INCREMENTAL."1000_MICRA_SELECTED" )
      Not()
      Move(in := #FC_NUMBER, out1 => "DB440_MACHINE_ALARM_DECODING".GLOBAL_ALARMS_MACHINE.WARNING_DECODING)
      wire#w1
      S_Coil( "DB440_MACHINE_ALARM_DECODING".ALARMS_CENTRAL.WARNING )
   END_RUNG
   RUNG wire#w1
      N_Trig( "DB2011_MODES_GENERAL_MG2".INCREMENTAL.WARNING_GONE )
      Move(in := 0, out1 => "DB440_MACHINE_ALARM_DECODING".GLOBAL_ALARMS_MACHINE.WARNING_DECODING)
      R_Coil( "DB440_MACHINE_ALARM_DECODING".ALARMS_CENTRAL.WARNING )
   END_RUNG
   // the same network as SCL:
   #_w1 := NOT (NOT "DB2011_MODES_GENERAL_MG2".INCREMENTAL.INCREMENTAL_MODE_SELECTED AND NOT "DB2011_MODES_GENERAL_MG2".INCREMENTAL."1_MICRA_SELECTED" AND NOT "DB2011_MODES_GENERAL_MG2".INCREMENTAL."10_MICRA_SELECTED" AND NOT "DB2011_MODES_GENERAL_MG2".INCREMENTAL."100_MICRA_SELECTED" AND NOT "DB2011_MODES_GENERAL_MG2".INCREMENTAL."1000_MICRA_SELECTED");
   IF #_w1 THEN
       "DB440_MACHINE_ALARM_DECODING".GLOBAL_ALARMS_MACHINE.WARNING_DECODING := #FC_NUMBER;
       "DB440_MACHINE_ALARM_DECODING".ALARMS_CENTRAL.WARNING := TRUE;
   END_IF;
   #_w2 := NOT #_w1 AND "DB2011_MODES_GENERAL_MG2".INCREMENTAL.WARNING_GONE;   // falling edge
   "DB2011_MODES_GENERAL_MG2".INCREMENTAL.WARNING_GONE := #_w1;
   IF #_w2 THEN
       "DB440_MACHINE_ALARM_DECODING".GLOBAL_ALARMS_MACHINE.WARNING_DECODING := 0;
       "DB440_MACHINE_ALARM_DECODING".ALARMS_CENTRAL.WARNING := FALSE;
   END_IF;
END_REGION

REGION Network 23: INCREMENTAL MODES GENERAL CONDITIONS HELP
   RUNG wire#powerrail
      I_Contact( "DB2011_MODES_GENERAL_MG2".INCREMENTAL."1_MICRA_REQUEST" )
      I_Contact( "DB2011_MODES_GENERAL_MG2".INCREMENTAL."10_MICRA_REQUEST" )
      I_Contact( "DB2011_MODES_GENERAL_MG2".INCREMENTAL."100_MICRA_REQUEST" )
      I_Contact( "DB2011_MODES_GENERAL_MG2".INCREMENTAL."1000_MICRA_REQUEST" )
      Not()
      I_Contact( "DB2011_MODES_GENERAL_MG2".INCREMENTAL.INCREMENTAL_MODES_GENERAL_CONDITIONS )
      Coil( "DB2011_MODES_GENERAL_MG2".INCREMENTAL.INCREMENTAL_MODES_GENERAL_CONDITIONS_HELP )
   END_RUNG
   // the same network as SCL:
   "DB2011_MODES_GENERAL_MG2".INCREMENTAL.INCREMENTAL_MODES_GENERAL_CONDITIONS_HELP := NOT (NOT "DB2011_MODES_GENERAL_MG2".INCREMENTAL."1_MICRA_REQUEST" AND NOT "DB2011_MODES_GENERAL_MG2".INCREMENTAL."10_MICRA_REQUEST" AND NOT "DB2011_MODES_GENERAL_MG2".INCREMENTAL."100_MICRA_REQUEST" AND NOT "DB2011_MODES_GENERAL_MG2".INCREMENTAL."1000_MICRA_REQUEST") AND NOT "DB2011_MODES_GENERAL_MG2".INCREMENTAL.INCREMENTAL_MODES_GENERAL_CONDITIONS;
END_REGION

REGION Network 24: INCREMENTAL MODES INITIAL CONDITIONS HELP
   RUNG wire#powerrail
      I_Contact( "DB2011_MODES_GENERAL_MG2".INCREMENTAL."1_MICRA_REQUEST" )
      I_Contact( "DB2011_MODES_GENERAL_MG2".INCREMENTAL."10_MICRA_REQUEST" )
      I_Contact( "DB2011_MODES_GENERAL_MG2".INCREMENTAL."100_MICRA_REQUEST" )
      I_Contact( "DB2011_MODES_GENERAL_MG2".INCREMENTAL."1000_MICRA_REQUEST" )
      Not()
      Contact( "DB2011_MODES_GENERAL_MG2".INCREMENTAL.INCREMENTAL_MODES_GENERAL_CONDITIONS )
      I_Contact( "DB2011_MODES_GENERAL_MG2".INCREMENTAL.INCREMENTAL_MODES_INITIAL_CONDITIONS )
      Coil( "DB2011_MODES_GENERAL_MG2".INCREMENTAL.INCREMENTAL_MODES_INITIAL_CONDITIONS_HELP )
   END_RUNG
   // the same network as SCL:
   "DB2011_MODES_GENERAL_MG2".INCREMENTAL.INCREMENTAL_MODES_INITIAL_CONDITIONS_HELP := NOT (NOT "DB2011_MODES_GENERAL_MG2".INCREMENTAL."1_MICRA_REQUEST" AND NOT "DB2011_MODES_GENERAL_MG2".INCREMENTAL."10_MICRA_REQUEST" AND NOT "DB2011_MODES_GENERAL_MG2".INCREMENTAL."100_MICRA_REQUEST" AND NOT "DB2011_MODES_GENERAL_MG2".INCREMENTAL."1000_MICRA_REQUEST") AND "DB2011_MODES_GENERAL_MG2".INCREMENTAL.INCREMENTAL_MODES_GENERAL_CONDITIONS AND NOT "DB2011_MODES_GENERAL_MG2".INCREMENTAL.INCREMENTAL_MODES_INITIAL_CONDITIONS;
END_REGION
END_FUNCTION
